TYPE Measurement_Event :
STRUCT
	
END_STRUCT
END_TYPE

(* stored: Version 1.1.0.1, ProductVersion 3.1.4024.12
   DUT Measurement_Event: Id {37dafad3-7e0d-459b-923b-8095747dd2c0} *)
